SUBAPPLICATION Ventilsteuerung_Uebung_034 (* Analog-Eingang auf PWM Ausgang *)
  (* Standard: 61499-2 *)
  (* Version 1.0, 2023-10-23, franz *)
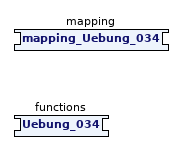
  SUBAPPS
    mapping : mapping_Uebung_034;
    functions : Uebung_034;
  END_SUBAPPS
END_SUBAPPLICATION
